// TIA Portal V20 export
TYPE "LGM_LKinCtrl_ControlNodeCommands"
// stored: Access Published
   STRUCT
      groupPower { ExternalAccessible := 'False'; ExternalVisible := 'False'; ExternalWritable := 'False'} : Bool;
      groupReset { ExternalAccessible := 'False'; ExternalVisible := 'False'; ExternalWritable := 'False'} : Bool;
      groupRestart : Array[1..7] of Bool;   // reinitialization of technology object
      groupHome { ExternalAccessible := 'False'; ExternalVisible := 'False'; ExternalWritable := 'False'} : Bool;
      selectedPath { ExternalAccessible := 'False'; ExternalVisible := 'False'; ExternalWritable := 'False'} : DInt;
      executeMovePath { ExternalAccessible := 'False'; ExternalVisible := 'False'; ExternalWritable := 'False'} : Bool;
      stopMovePath { ExternalAccessible := 'False'; ExternalVisible := 'False'; ExternalWritable := 'False'} : Bool;
      interruptMovePath { ExternalAccessible := 'False'; ExternalVisible := 'False'; ExternalWritable := 'False'} : Bool;
      resetMovePath { ExternalAccessible := 'False'; ExternalVisible := 'False'; ExternalWritable := 'False'} : Bool;
      abortMeasurementCmd { ExternalAccessible := 'False'; ExternalVisible := 'False'; ExternalWritable := 'False'} : Bool;
      setFlags { ExternalAccessible := 'False'; ExternalVisible := 'False'; ExternalWritable := 'False'} : Array[0.."LKINCTRL_NO_OF_LAST_SETFLAG"] of Bool;
      valueFlags { ExternalAccessible := 'False'; ExternalVisible := 'False'; ExternalWritable := 'False'} : Array[0.."LKINCTRL_NO_OF_LAST_VALUEFLAG"] of LReal;
      hmiLogic : Struct
         enable : Bool := TRUE;   // TRUE: Enable functionality of FB
         eStopActive : Bool;   // TRUE: EStop is active. TeachKinematics is blocked.
         motionEnable : Bool := true;   // TRUE: Motion is allowed, FALSE: Motion is not allowed.
         externalInterlock { ExternalVisible := 'False'; ExternalWritable := 'False'} : Bool := false;   // Generic external lock to block HMI.
         externalManualOverride { ExternalVisible := 'False'; ExternalWritable := 'False'} : Int := -1;   // Optional external manual override.
         infeedEnabled : Bool := true;   // Enable feedback from the infeed.
         infeedError : Bool := false;   // Error feedback from the infeed.
         axesCouplingEnabled : Bool := true;   // Enable feedback from the axes coupling.
      END_STRUCT;
   END_STRUCT;
   // setFlags[0] := TRUE;
   // setFlags[1] := FALSE;
   // setFlags[2..3] := TRUE;
   // setFlags[4..30] := FALSE;
   // valueFlags[0..30] := 0.0;
END_TYPE
